{attribute 'GeneratedUsingTerminal: EK1100-0000-0018'}
{attribute addProperty BoxType "EK1100-0000-0018"}
{attribute addProperty Id "Beckhoff_EPP5xxxEK1122Beckhoff_EPP5xxxEK1122_EF1F281E304"}
{attribute addProperty CRC "3469417631"}
{attribute addProperty Size "304"}
TYPE Beckhoff_EPP5xxx_CECB1C9F EXTENDS EK1100_1FC0878B :
STRUCT
	{attribute addProperty Name "Beckhoff_EPP5xxxEK1122"}
	Beckhoff_EPP5xxxEK1122 : Beckhoff_EPP5xxxEK1122_EF1F281E;
END_STRUCT
END_TYPE

(* stored: Version 1.2.0.0, ProductVersion 3.1.4024.9
   DUT Beckhoff_EPP5xxx_CECB1C9F: Id {6e9dd16c-443d-46e2-9107-58e9207ae43b} *)
